FUNCTION_BLOCK FB_ShippingArea EXTENDS FB_ModeBase_V2 IMPLEMENTS I_UnitState
VAR_INPUT
	FanucRobot 		: REFERENCE TO FB_FanucRobot_Basic_V2;
	Service 		: REFERENCE TO ST_ShippingService;
	INPUT       	: REFERENCE TO ST_InputTable;
	OUTPUT			: REFERENCE TO ST_OutputTable;
	Motor    		: REFERENCE TO UNI_MotorList;
    Reset           : REFERENCE TO BOOL;
	Stop 			: REFERENCE TO BOOL;
    bStopMem 		: REFERENCE TO BOOL;
END_VAR
VAR_OUTPUT
	Homed : BOOL;
	RobotResetCMD : BOOL;
END_VAR
VAR
	abort	: BOOL;

	// 連動暫停 - 任一 Service 錯誤時暫停所有其他 Service
	_bAnyServiceError : BOOL;

	//Machine Service
	fbShippingHoming 				: FB_ShippingHoming;
	
	// Same / Difference CV Service
	fbShippingRobot_TransmitCVEnd :	FB_ShippingRobot_TransmitCVEnd;

	//Robot Service
	fbShippingRobot_Left 			: FB_ShippingRobot_Left;
	fbShippingRobot_Right 			: FB_ShippingRobot_Right;
	
	//HansLaser HandShake TransCV Service
	fbShippingLeftSideTransCV		: FB_ShippingTransCV_LeftSide;
	fbShippingRightSideTransCV		: FB_ShippingTransCV_RightSide;
END_VAR

SUPER^();

IF __ISVALIDREF(PackTag) THEN
    eModeCommand  := PackTag.Command.UnitMode;
    eStateCommand := PackTag.Command.CntrlCmd;
ELSE
    RETURN;
END_IF

ACTION A00_Service:
// ============================================================================
// 連動暫停邏輯 - 任一 Service 錯誤時，暫停所有其他 Service
// ============================================================================
_bAnyServiceError :=
	Service.AutoMode_ShippingRobot_TransmitCVEnd.Status.Error OR
	Service.AutoMode_ShippingRobot_Left.Status.Error OR
	Service.AutoMode_ShippingRobot_Right.Status.Error OR
	Service.AutoMode_ShippingTransCV_LeftSide.Status.Error OR
	Service.AutoMode_ShippingTransCV_RightSide.Status.Error;

fbShippingRobot_TransmitCVEnd(
	Execute:= Service.AutoMode_ShippingRobot_TransmitCVEnd.Command.Execute,
	Abort:= Service.AutoMode_ShippingRobot_TransmitCVEnd.Command.Abort OR THIS^.Abort OR _bAnyServiceError,
	Reset:= Reset, 
	ObjectName:= 'Shipping Fanuc Robot TransmitCVEnd', 
	INPUT:=INPUT,
	Motor :=Motor,
	Busy=> Service.AutoMode_ShippingRobot_TransmitCVEnd.Status.Busy, 
	Done=> Service.AutoMode_ShippingRobot_TransmitCVEnd.Status.Done, 
	Aborted=> , 
	Error=> Service.AutoMode_ShippingRobot_TransmitCVEnd.Status.Error, 
	ErrorID=> , 
	Status=> Service.AutoMode_ShippingRobot_TransmitCVEnd.Status.Status, 
	UniqueErrorCode=> , 
	Robot:= FanucRobot, 
	Info:= Service.AutoMode_ShippingRobot_TransmitCVEnd.Info, 
	Stop:= bStopMem,
	fbSHippingHomingBusy := fbShippingHoming.xBusy);
	
fbShippingRobot_Left(
	Execute:= service.AutoMode_ShippingRobot_Left.Command.Execute,
	Abort:= Service.AutoMode_ShippingRobot_Left.Command.Abort OR THIS^.Abort OR _bAnyServiceError,
	Reset:= Reset,
	ObjectName:= 'Shipping Fanuc Robot Left', 
	Busy=> Service.AutoMode_ShippingRobot_Left.Status.Busy, 
	Done=> Service.AutoMode_ShippingRobot_Left.Status.Done, 
	Aborted=> , 
	Error=> Service.AutoMode_ShippingRobot_Left.Status.Error, 
	ErrorID=> , 
	Status=> Service.AutoMode_ShippingRobot_Left.Status.Status, 
	UniqueErrorCode=> , 
	Robot:= FanucRobot, 
	Info:= Service.AutoMode_ShippingRobot_Left.Info, 
	Stop:=bStopMem,
	Buzz := DAS_CoreSys.MachineControl._Buzz,
	RedLamp:= DAS_CoreSys.MachineControl._RedLamp,
	bCompleteRequest := Service.AutoMode_ShippingRobot_Left.bCompleteRequest,
	bTransCVInPosition => Service.AutoMode_ShippingRobot_Left.bTransCVInPosition,
	Input := INPUT);
	
fbShippingRobot_Right(
	Execute:= Service.AutoMode_ShippingRobot_Right.Command.Execute,
	Abort:= Service.AutoMode_ShippingRobot_Right.Command.Abort OR THIS^.Abort OR _bAnyServiceError,
	Reset:= Reset,
	ObjectName:= 'Shipping Fanuc Robot Right', 
	Busy=> Service.AutoMode_ShippingRobot_Right.Status.Busy, 
	Done=> Service.AutoMode_ShippingRobot_Right.Status.Done, 
	Aborted=> , 
	Error=> Service.AutoMode_ShippingRobot_Right.Status.Error, 
	ErrorID=> , 
	Status=> Service.AutoMode_ShippingRobot_Right.Status.Status, 
	UniqueErrorCode=> , 
	Robot:= FanucRobot, 
	Info:= Service.AutoMode_ShippingRobot_Right.Info, 
	Stop:= bStopMem,
	Buzz := DAS_CoreSys.MachineControl._Buzz,
	RedLamp:= DAS_CoreSys.MachineControl._RedLamp,
	bCompleteRequest := Service.AutoMode_ShippingRobot_Right.bCompleteRequest,
	bTransCVInPosition => Service.AutoMode_ShippingRobot_Right.bTransCVInPosition,
	Input := INPUT);
	
fbShippingHoming(
	xDone=> ,
	xBusy=> ,
	xError=> ,
	xExecute:= ,
	xAbort:= _bAnyServiceError,
	FanucRobot:= FanucRobot, 
	Homed:= Homed, 
	xAborted=> , 
	iErrorID=> , 
	ErrorMsg=> , 
	RobotResetCMD=> RobotResetCMD,
	Service := Service,
	input := INPUT,
	Output := OUTPUT,
	Motor := Motor);
	
fbShippingLeftSideTransCV(
	xDone=> Service.AutoMode_ShippingTransCV_LeftSide.Status.Done,
	xBusy=> Service.AutoMode_ShippingTransCV_LeftSide.Status.Busy,
	xError=> Service.AutoMode_ShippingTransCV_LeftSide.Status.Error,
	xExecute:= Service.AutoMode_ShippingTransCV_LeftSide.Command.Execute,
	xAbort:= Service.AutoMode_ShippingTransCV_LeftSide.Command.Abort OR THIS^.abort OR _bAnyServiceError,
	xReset:= Service.AutoMode_ShippingTransCV_LeftSide.Command.Reset,
	Cylinder:= , 
	TimeOut:= , 
	Input:= input, 
	OutPut:= output, 
	Motor:= , 
	ShippingTransCVRequest_LeftSide:= Service.AutoMode_ShippingTransCV_LeftSide.ShippingTransCVRequest_LeftSide, 
	RobotStatus:= Service.AutoMode_ShippingRobot_Left.Status, 
	xAborted=> , 
	iErrorID=> , 
	ErrorMsg=> Service.AutoMode_ShippingTransCV_LeftSide.Status.Status);
	
fbShippingRightSideTransCV(
	xDone=> Service.AutoMode_ShippingTransCV_RightSide.Status.Done,
	xBusy=> Service.AutoMode_ShippingTransCV_RightSide.Status.Busy,
	xError=> Service.AutoMode_ShippingTransCV_RightSide.Status.Error,
	xExecute:= Service.AutoMode_ShippingTransCV_RightSide.Command.Execute,
	xAbort:= Service.AutoMode_ShippingTransCV_RightSide.Command.Abort OR THIS^.abort OR _bAnyServiceError,
	xReset:= Service.AutoMode_ShippingTransCV_RightSide.Command.Reset,
	Cylinder:= , 
	TimeOut:= , 
	Input:= input, 
	OutPut:= output, 
	Motor:= , 
	ShippingTransCVRequest_RightSide:= Service.AutoMode_ShippingTransCV_RightSide.ShippingTransCVRequest_RightSide, 
	RobotStatus:= Service.AutoMode_ShippingRobot_Right.Status, 
	xAborted=> , 
	iErrorID=> , 
	ErrorMsg=> Service.AutoMode_ShippingTransCV_RightSide.Status.Status);
END_ACTION

METHOD M_Aborted
abort := false;
M_StateComplete();
END_METHOD

METHOD M_Aborting
abort := true;
M_StateComplete();
END_METHOD

METHOD M_Clearing
M_StateComplete();
END_METHOD

METHOD M_Complete
M_StateComplete();
END_METHOD

METHOD M_Completing
M_StateComplete();
END_METHOD

METHOD M_Execute
CASE eModeCurrent OF
	E_UnitMode.Manual:
		;
	E_UnitMode.Auto:
		;
END_CASE
A00_Service();
//M_StateComplete();
END_METHOD

METHOD M_Held
M_StateComplete();
END_METHOD

METHOD M_Holding
M_StateComplete();
END_METHOD

METHOD M_Idle
M_StateComplete();
END_METHOD

METHOD M_Resetting
M_StateComplete();
END_METHOD

METHOD M_StartHoming
VAR_INPUT
END_VAR
fbShippingHoming.xExecute := TRUE;
END_METHOD

METHOD M_Starting
M_StateComplete();
END_METHOD

METHOD M_StopHoming
VAR_INPUT
END_VAR
fbShippingHoming.xExecute := False;
END_METHOD

METHOD M_Stopped
M_StateComplete();
END_METHOD

METHOD M_Stopping
M_StateComplete();
END_METHOD

METHOD M_Suspended
M_StateComplete();
END_METHOD

METHOD M_Suspending
M_StateComplete();
END_METHOD

METHOD M_Undefined
M_StateComplete();
END_METHOD

METHOD M_Unholding
M_StateComplete();
END_METHOD

METHOD M_Unsuspending
M_StateComplete();
END_METHOD

END_FUNCTION_BLOCK

(* stored: Version 1.1.0.1, ProductVersion 3.1.4024.13
   POU FB_ShippingArea: Id {48d05f6d-623d-41de-9852-ec870669682f}, SpecialFunc None
   Folder States: Id {f81533be-596c-4ef2-b789-36286d227524}
   Action A00_Service: Id {d3e5687a-8989-4023-9d99-a9d8ba12dedd}
   Method M_Aborted: Id {3b7aeb74-3c46-4095-9c8f-17f92de17ccd}
   Method M_Aborting: Id {e034d6b1-5633-4f6c-ba14-3db2cdadef3b}
   Method M_Clearing: Id {51942349-3aa5-4126-9672-95e7ba2cdf88}
   Method M_Complete: Id {0a50b301-c693-48df-b8ab-0efb990f6cc3}
   Method M_Completing: Id {e68e890d-8f79-49c6-9fe0-29fa071f049c}
   Method M_Execute: Id {105523e7-c49e-464d-8a47-e74c9b948053}
   Method M_Held: Id {a2428c09-a67e-40ee-a6c4-ea9fff4dfdc1}
   Method M_Holding: Id {1f3ecc8d-4af4-4df5-ab43-b5172564f883}
   Method M_Idle: Id {39d99d48-42ad-4845-b0e8-0ccf860df6c2}
   Method M_Resetting: Id {933d9293-477d-4616-861c-b8157948a9f8}
   Method M_StartHoming: Id {15fc3ed6-f365-4832-a7b5-c735e9e105f3}
   Method M_Starting: Id {2e9f53da-22f0-4ad6-856d-87f17da6dc0f}
   Method M_StopHoming: Id {5665e39d-7e26-4fbf-b1d0-3b763074b645}
   Method M_Stopped: Id {db54aee9-82dc-4e05-949c-2853586d3c03}
   Method M_Stopping: Id {9b99ea87-8833-48c9-81cb-4c0516bf33e3}
   Method M_Suspended: Id {59654d4a-727d-4de9-9547-06d1cc9abbc0}
   Method M_Suspending: Id {4599f32f-9426-4e3a-80c1-6199d77adedc}
   Method M_Undefined: Id {33a8122a-be5c-4f80-90a6-433b9df1dea4}
   Method M_Unholding: Id {9f10015f-fd10-4150-8900-f7bbf2fdb92b}
   Method M_Unsuspending: Id {3eb01f5b-faa2-481b-8df8-a76484441fac} *)
